{attribute 'GeneratedUsingTerminal: EL5101-0000-0001'}
{attribute addProperty BoxType "EL5101-0000-0001"}
{attribute addProperty Id "InputsAT %I*Inputs_B90637B95OutputsAT %Q*Outputs_C6781B153WcStateAT %I*WcState_9091E0EB2InfoDataAT %I*InfoData_94A18F5E2"}
{attribute addProperty CRC "2787048877"}
{attribute addProperty Size "12"}
TYPE EL5101_A61EFDAD EXTENDS EtcSlaveTerminalBase_947E5A46 :
STRUCT
	{attribute addProperty Name "Inputs"}
	Inputs : Inputs_B90637B9;
	{attribute addProperty Name "Outputs"}
	Outputs : Outputs_C6781B15;
	{attribute addProperty Name "WcState"}
	WcState : WcState_9091E0EB;
	{attribute addProperty Name "InfoData"}
	InfoData : InfoData_94A18F5E;
END_STRUCT
END_TYPE

(* stored: Version 1.2.0.0, ProductVersion 3.1.4024.9
   DUT EL5101_A61EFDAD: Id {4b8607c8-1d53-42a6-88a6-8a914a42c94c} *)
